FUNCTION_BLOCK E_R_TRIG
  {SET_ATTRIBUTE(OpcUa, Service)}
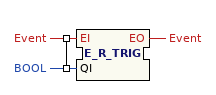
  EVENT_INPUT
    EI WITH QI;
  END_EVENT
  EVENT_OUTPUT
    EO;
  END_EVENT
  VAR_INPUT
    QI : BOOL; {SET_ATTRIBUTE(OpcUa, Variable.RUN)}
  END_VAR
END_FUNCTION_BLOCK
